{attribute 'linkalways'} 
{attribute 'no_explicit_call' := 'This FB is a CLASS and must be accessed using methods or properties'}
{attribute 'enable_dynamic_creation'}
FUNCTION_BLOCK HomeCommand EXTENDS Mc2Command
VAR
	fb : Tc2_Mc2.Mc_Home;
END_VAR

METHOD PUBLIC CyclicCall
SUPER^.CyclicCall();
fb(Axis := axis_ref);
END_METHOD

(*FB_Init is always available implicitly and it is used primarily for initialization.
The return value is not evaluated. For a specific influence, you can also declare the
methods explicitly and provide additional code there with the standard initialization
code. You can evaluate the return value.*)
METHOD FB_Init : BOOL
VAR_INPUT
	(* TRUE: the retain variables are initialized (reset warm / reset cold)*)
	bInitRetains : BOOL;
	(* TRUE: the instance will be copied to the copy code afterward (online change)*)
	bInCopyCode	: BOOL;
	axis : Axis;
	position : LREAL := Tc2_Mc2.Default_Home_Position;
	homing_mode : HomingMode := HomingMode.Default;
	buffer_mode	: MotionBufferMode := MotionBufferMode.Aborting;
END_VAR
fb.Position := position;
fb.HomingMode := Mc2HomingModeConvertTo(homing_mode);
fb.BufferMode := Mc2BufferModeConvertTo(buffer_mode);
END_METHOD

METHOD PROTECTED OnExecuting
VAR_INPUT
	state_control : AsyncCommandStateControl;
END_VAR
fb.Execute := TRUE;

IF fb.Done THEN
	state_control.Next();
	fb.Execute := FALSE;
END_IF

IF fb.CommandAborted THEN
	Abort();
	fb.Execute := FALSE;
END_IF

IF fb.Error THEN
	state_control.Error(fb.ErrorId);
	fb.Execute := FALSE;
END_IF
END_METHOD

END_FUNCTION_BLOCK

(* stored: Version 1.1.0.1
   POU HomeCommand: Id {517256b3-8391-4233-9af6-0bb5e27e1fcd}, SpecialFunc None
   Method CyclicCall: Id {31bbba72-1e8e-47ee-8a66-552d86497abf}
   Method FB_Init: Id {e4e46bb4-bea9-4312-9329-19efff41832f}
   Method OnExecuting: Id {9508e2de-9d28-425c-b0a6-3b92a2a5ba7b} *)
